{attribute 'qualified_only'}
VAR_GLOBAL
	bM1Motor		:BOOL; // M2 motor 
	bM2Motor 		:BOOL;	//M2 Motor
END_VAR

(* stored: Version 1.1.0.1, ProductVersion 3.1.4024.12
   GVL output: Id {c7dcf864-6141-4728-8cb4-8f4d99090033} *)
